FUNCTION_BLOCK FB_SealBar EXTENDS FB_ComponentBase
VAR
    // Data
    _SetTemperature    : LREAL;
    _ActualTemperature : LREAL;

    // IO
    _Heat AT %Q* : BOOL;

    // Other items
    TempUpdate   : TON;
    _InTempRange : BOOL;
END_VAR

PROPERTY ActualTemperature : LREAL
GET
ActualTemperature := _ActualTemperature;
END_GET
END_PROPERTY

METHOD CyclicLogic
VAR_INPUT
END_VAR
IF NOT _InitComplete THEN
    _InitComplete := Initialize();
    RETURN;
END_IF

SUPER^.CyclicLogic();

//Read data from Parameters

/// Set from the property SetTemperature := _Param[SETTEMP].Value;

(*Temperature for simulation of temperature changes
This will add 0.3 every 100ms to actual until it gets to Setpoint
It will subtract 0.1 degrees every 100ms unitl it is down to setpoint or 20
Do not set below 20 or it will not get passed resetting*)
TempUpdate(IN := NOT TempUpdate.Q, PT := T#100MS);
IF TempUpdate.Q THEN
    IF _Heat AND _ActualTemperature < _SetTemperature THEN
        _ActualTemperature := _ActualTemperature + 0.3;
    ELSIF _ActualTemperature > 20 THEN
        _ActualTemperature := _ActualTemperature - 0.1;
    END_IF
END_IF

IF ABS(_SetTemperature - _ActualTemperature) < 1 THEN
    _InTempRange := TRUE;
ELSE
    _InTempRange := FALSE;
END_IF
END_METHOD

PROPERTY Heat : BOOL
GET
Heat := _Heat;
END_GET
SET
_Heat := Heat;
END_SET
END_PROPERTY

PROPERTY InTempRange : BOOL
GET
InTempRange := _InTempRange;
END_GET
END_PROPERTY

PROPERTY SetTemperature : LREAL
GET
SetTemperature := _SetTemperature;
END_GET
SET
_SetTemperature := SetTemperature;
END_SET
END_PROPERTY

END_FUNCTION_BLOCK

(* stored: Version 1.1.0.1
   POU FB_SealBar: Id {ab562724-f2ca-416e-b831-b15d6083aa70}, SpecialFunc None
   Folder I_ComponentBase: Id {6988ed05-0623-4392-a74b-659338262400}
   Folder I_CyclicFB: Id {9c7dbd40-2329-4d37-80bb-9312e30eceba}
   Folder I_SealBar: Id {6692dfd2-b960-4d90-9dce-e743cce28a6f}
   Property ActualTemperature: Id {2c1e9d11-f43f-485b-999d-29733c4a40cc}
   Get Get: Id {825b3faf-f9d0-4280-92a0-347a6febd8aa}
   Method CyclicLogic: Id {2eb5b232-4650-451a-acea-d277a3303acf}
   Property Heat: Id {7e9e9463-3cab-4a5f-b56e-58ed71a977eb}
   Get Get: Id {3bf52207-ca86-44c6-bad6-49d059e34aa5}
   Set Set: Id {0b515c20-43d3-4d3a-b294-c24de8301402}
   Property InTempRange: Id {ef285aec-9753-486c-bd66-9094bbe2910e}
   Get Get: Id {43492085-da08-4922-9e03-47515fde9ff0}
   Property SetTemperature: Id {b0235246-fc0d-416e-ad23-71c3fcb36431}
   Get Get: Id {adca20c1-327b-458b-93a9-e53da43a8d1c}
   Set Set: Id {5eabeff8-a172-4183-a5e1-15e3ae65271e} *)
